// TIA Portal V15.1 export
// export: Created 2022-12-21T11:46:37.002822Z, ExportSettings None
FUNCTION_BLOCK "test"   // FB, FBD
TITLE = test
{ S7_Optimized_Access := 'TRUE' }
// test description
// stored: AutoNumber true, MemoryReserve 100
   VAR
      Mode : "Mode_PLC_FB";   // Mode
   END_VAR
BEGIN

REGION Network 1: test_network
   // test_network_description
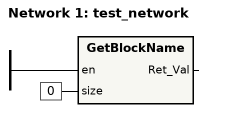
   GetBlockName(size := 0);
END_REGION
END_FUNCTION_BLOCK
